(* IEC 61131-3 sources: AQUA-FLOW-System/Source_Code, 3 files *)

(* ---- GVL_Tank.st ---- *)
{attribute 'qualified_only'}
VAR_GLOBAL
    // ============================================================
    // 1. INPUTS (HMI Pushbuttons & Physical Control Panel Switches)
    // ============================================================
    xStartButton        : BOOL;     // System Start / Resume command
    xStopButton         : BOOL;     // System Stop command (Normal shutdown)
    xHoldButton         : BOOL;     // System Pause / Hold command
    xEmStop             : BOOL;     // Emergency Stop physical input (NC contact)
    xEmStop_Latched     : BOOL;     // Latched Emergency Stop state (Requires reset)
    xAutoModeButton     : BOOL;     // HMI pushbutton for Auto mode selection
    xManualModeButton   : BOOL;     // HMI pushbutton for Manual mode selection

    xResetButton        : BOOL;     // Fault / Alarm Reset command (HMI or Physical)
    xAlarmTrip          : BOOL;     // Latched System Fault state (Locks system)

    xSelectorSwitch     : BOOL;     // HMI Mode Selector Switch (FALSE = Manual, TRUE = Auto)

    // ============================================================
    // 2. MANUAL CONTROLS (Direct Actuator Overrides in Manual Mode)
    // ============================================================
    xManualInlet        : BOOL;     // Manual command to open inlet valve
    xManualOutlet       : BOOL;     // Manual command to run outlet pump

    // ============================================================
    // 3. PROCESS VARIABLES (Analog & Continuous Data)
    // ============================================================
    rTankLevel          : REAL;     // Current tank water level (Scaled: 0.0 - 100.0 %)

    // ============================================================
    // 4. OUTPUTS (Physical Hardware Control Signals)
    // ============================================================
    xInletValve         : BOOL;     // Inlet Valve command (TRUE = Open)
    xOutletPump         : BOOL;     // Outlet Pump command (TRUE = Run)

    // ============================================================
    // 5. SYSTEM STATUS & ALARMS (HMI Indicators & SCADA Integration)
    // ============================================================
    xSystemRunning      : BOOL;     // System is currently active and executing sequence
    xSystemHold         : BOOL;     // System is temporarily paused (Hold state)
    xLevelAlarm         : BOOL;     // Critical level alarm trigger (Tank < 5% or > 95%)

    xAutoModeActive     : BOOL;     // Active control mode feedback flag: Auto
    xManualModeActive   : BOOL;     // Active control mode feedback flag: Manual

    // Hardware Interlocks (Failsafe Sensors)
    xHighFloatSwitch    : BOOL;     // High-Level Hardware Interlock (TRUE = Overflow risk)
    xLowFloatSwitch     : BOOL;     // Low-Level Hardware Interlock (TRUE = Pump dry-run risk)

    iCycleCount         : INT := 0; // Accumulated water draining cycles counter

    sStatusText         : STRING;   // Current system state message for HMI display

    // ============================================================
    // 6. INDICATOR LAMPS (Control Panel Status Lights)
    // ============================================================
    xLamp_Red           : BOOL;     // Red light (System Fault / Alarm Active)
    xLamp_Yellow        : BOOL;     // Yellow light (System in Standby / Manual Mode)
    xLamp_Green         : BOOL;     // Green light (System Running normally in Auto)
END_VAR

(* ---- FB_Simulation.st ---- *)
FUNCTION_BLOCK FB_Simulation
VAR_INPUT
    xInletOpen  : BOOL;
    xOutletRun  : BOOL;
END_VAR
VAR_IN_OUT
    rLevel      : REAL;
END_VAR
VAR
    fbTimer     : TON;
    xTrigger    : BOOL;
END_VAR
/////////////////////////////
(* ==========================================================
   Water Tank Behavior Simulator Block - FIXED
   ========================================================== *)

// Generate a continuous 100ms pulse for the simulation step
fbTimer(IN := NOT xTrigger, PT := T#100MS);

// Create a 1-scan-cycle trigger when the timer completes
IF fbTimer.Q THEN
    xTrigger := TRUE;
ELSE
    xTrigger := FALSE;
END_IF;

// Execute level calculations only when the trigger is active
IF xTrigger THEN

    // 1. Simulation: Filling Phase (Inlet Open, Pump Stopped)
    IF xInletOpen AND NOT xOutletRun THEN
        IF rLevel < 100.0 THEN
            rLevel := rLevel + 0.5; // Increase level by 0.5% per 100ms
        END_IF
    END_IF

    // 2. Simulation: Draining Phase (Pump Running, Inlet Closed)
    IF xOutletRun AND NOT xInletOpen THEN
        IF rLevel > 0.0 THEN
            rLevel := rLevel - 0.8; // Decrease level by 0.8% per 100ms
        END_IF
    END_IF

    // 3. Simulation: Simultaneous Operation (Both Active)
    IF xInletOpen AND xOutletRun THEN
        IF rLevel < 100.0 AND rLevel > 0.0 THEN
            rLevel := rLevel - 0.3; // Net decrease (Draining rate > Filling rate)
        END_IF
    END_IF

    // 4. Boundary Protection (Clamp values to prevent out-of-bounds)
    IF rLevel > 100.0 THEN
        rLevel := 100.0;
    ELSIF rLevel < 0.0 THEN
        rLevel := 0.0;
    END_IF

END_IF

(* ---- FB_TankLogic_Updated.st ---- *)
FUNCTION_BLOCK FB_TankLogic_Updated
VAR_INPUT

END_VAR
VAR_OUTPUT
END_VAR
VAR
    iState : INT := 0;
END_VAR
////////////////////////////
// ==========================================================
// 1. Mode Selection & Safety Latching
// ==========================================================
// Map physical/HMI selector switch to internal mode flags
GVL_Tank.xAutoModeActive   := GVL_Tank.xSelectorSwitch;
GVL_Tank.xManualModeActive := NOT GVL_Tank.xSelectorSwitch;

// --- E-STOP Latching Logic ---
// Immediately latch the E-Stop state upon activation to prevent accidental restart
IF GVL_Tank.xEmStop THEN
    GVL_Tank.xEmStop_Latched := TRUE;
END_IF

// Unlatch E-Stop only if the physical button is released (pulled up) AND the operator issues a Reset command
IF GVL_Tank.xResetButton AND NOT GVL_Tank.xEmStop THEN
    GVL_Tank.xEmStop_Latched := FALSE;
END_IF

// ==========================================================
// 2. Alarm Management
// ==========================================================
// 2.1 Detect and latch critical process alarms (Overflow or Dry-run conditions)
IF (GVL_Tank.rTankLevel > 95.0) OR GVL_Tank.xHighFloatSwitch OR GVL_Tank.xLowFloatSwitch THEN
    GVL_Tank.xLevelAlarm := TRUE;
    GVL_Tank.xAlarmTrip  := TRUE;
ELSE
    GVL_Tank.xLevelAlarm := FALSE;
END_IF

// 2.2 Acknowledge and clear alarms only when process values return to safe boundaries and a Reset is triggered
IF GVL_Tank.xResetButton AND (GVL_Tank.rTankLevel <= 95.0) AND NOT GVL_Tank.xHighFloatSwitch AND NOT GVL_Tank.xLowFloatSwitch THEN
    GVL_Tank.xAlarmTrip := FALSE;
END_IF

// ==========================================================
// 3. Safety Interlock State Management
// ==========================================================
// Force the sequence state machine back to initialization (State 0) if the system is halted or E-Stop is active
IF NOT GVL_Tank.xSystemRunning OR GVL_Tank.xEmStop_Latched THEN
    iState := 0;
END_IF

// ==========================================================
// 4. Auto / Manual / Standby Control
// ==========================================================
// ------------------------------------------------------
// 4.1 Auto Mode Sequence
// ------------------------------------------------------
IF GVL_Tank.xAutoModeActive AND NOT GVL_Tank.xSystemHold AND NOT GVL_Tank.xAlarmTrip AND NOT GVL_Tank.xEmStop_Latched THEN

    // Sequence progression based on tank level thresholds
    IF GVL_Tank.rTankLevel <= 20.0 THEN
        iState := 1;     // Transition to Filling Phase
    ELSIF GVL_Tank.rTankLevel >= 80.0 THEN
        IF iState = 1 THEN
            GVL_Tank.iCycleCount := GVL_Tank.iCycleCount + 1; // Increment cycle counter upon fill completion
        END_IF
        iState := 2;     // Transition to Draining Phase
    ELSIF iState = 0 THEN
        iState := 1;     // Initial Startup Phase
    END_IF

    // Actuator control mapped to current sequence state
    IF iState = 1 THEN
        GVL_Tank.xInletValve := TRUE;
        GVL_Tank.xOutletPump := FALSE;
    ELSIF iState = 2 THEN
        GVL_Tank.xInletValve := FALSE;
        GVL_Tank.xOutletPump := TRUE;
    END_IF

// ------------------------------------------------------
// 4.2 Manual Mode Override
// ------------------------------------------------------
ELSIF GVL_Tank.xManualModeActive AND NOT GVL_Tank.xEmStop_Latched THEN

    iState := 0; // Override and reset Auto sequence state

    // Mutual exclusion interlock: Prevent simultaneous opening of inlet and outlet to avoid hydraulic bypass
    IF GVL_Tank.xManualInlet AND GVL_Tank.xManualOutlet THEN
        GVL_Tank.xInletValve := FALSE;
        GVL_Tank.xOutletPump := FALSE;
    ELSE
        GVL_Tank.xInletValve := GVL_Tank.xManualInlet;
        GVL_Tank.xOutletPump := GVL_Tank.xManualOutlet;
    END_IF

// ------------------------------------------------------
// 4.3 Standby / Idle Mode
// ------------------------------------------------------
ELSE
    // Ensure all actuators are safely de-energized
    GVL_Tank.xInletValve := FALSE;
    GVL_Tank.xOutletPump := FALSE;
    iState := 0;
END_IF

// ==========================================================
// 5. Status Message Display (Priority Routing)
// ==========================================================
// Prioritized HMI messaging pipeline (Highest priority conditions overwrite lower ones)
IF GVL_Tank.xEmStop_Latched THEN
    GVL_Tank.sStatusText := 'EMERGENCY STOP ACTIVATED!';
ELSIF GVL_Tank.xAlarmTrip THEN
    GVL_Tank.sStatusText := 'SYSTEM FAULT (ALARM)';
ELSIF (GVL_Tank.rTankLevel <= 0.0) AND GVL_Tank.xManualOutlet THEN
    GVL_Tank.sStatusText := 'WARNING: TANK EMPTY (DRY-RUN)';
ELSIF (GVL_Tank.rTankLevel >= 95.0) AND GVL_Tank.xManualInlet THEN
    GVL_Tank.sStatusText := 'WARNING: TANK FULL (OVERFLOW)';
ELSIF iState = 1 THEN
    GVL_Tank.sStatusText := 'FILLING WATER';
ELSIF iState = 2 THEN
    GVL_Tank.sStatusText := 'DRAINING WATER';
ELSE
    GVL_Tank.sStatusText := 'STANDBY';
END_IF

// ==========================================================
// 6. Control Panel Indicator Lamps
// ==========================================================
// Red: Active when an alarm is tripped or E-Stop is engaged
GVL_Tank.xLamp_Red    := GVL_Tank.xAlarmTrip OR GVL_Tank.xEmStop_Latched;

// Yellow: Active when the system is not running or switched to Manual mode
GVL_Tank.xLamp_Yellow := (NOT GVL_Tank.xSystemRunning) OR GVL_Tank.xManualModeActive;

// Green: Active only when the system is running smoothly in Auto mode with no faults
GVL_Tank.xLamp_Green  := GVL_Tank.xSystemRunning AND GVL_Tank.xAutoModeActive AND NOT GVL_Tank.xAlarmTrip AND NOT GVL_Tank.xEmStop_Latched;

// ==========================================================
// 7. Process Hardware Protection (End-of-scan Override)
// ==========================================================
// Absolute hardware override at the end of the scan cycle (Failsafe execution)
IF NOT GVL_Tank.xSystemRunning OR GVL_Tank.xEmStop_Latched THEN
    GVL_Tank.xInletValve := FALSE;
    GVL_Tank.xOutletPump := FALSE;
END_IF

// Prevent tank overflow regardless of active control mode
IF (GVL_Tank.rTankLevel >= 95.0) OR GVL_Tank.xHighFloatSwitch THEN
    GVL_Tank.xInletValve := FALSE;
END_IF

// Prevent pump dry-run cavitation regardless of active control mode
IF (GVL_Tank.rTankLevel <= 0.0) OR GVL_Tank.xLowFloatSwitch THEN
    GVL_Tank.xOutletPump := FALSE;
END_IF
